// TwinCAT 3 PLC project OEF_1
// ProgramVersion: 3.1.4024.0
// libraries:
//   Tc2_Standard, * (Beckhoff Automation GmbH)
//   Tc2_System, * (Beckhoff Automation GmbH)
//   Tc3_Module, * (Beckhoff Automation GmbH)
// project tree:
//   / PlcTask.TcTTO
//   POUs/ MAIN.TcPOU
// real-time tasks:
//   TASK PlcTask: cycle T#10ms, priority 20, ADS port 350
//   TASK PlcTask1: cycle T#10ms, priority 21, ADS port 351
//   TASK PlcTask2: cycle T#10ms, priority 22, ADS port 352
//   TASK PlcTask3: cycle T#10ms, priority 23, ADS port 353
//   TASK PlcTask4: cycle T#10ms, priority 24, ADS port 354
//   TASK PlcTask5: cycle T#10ms, priority 25, ADS port 355
//   TASK PlcTask6: cycle T#10ms, priority 26, ADS port 356
// I/O:
//   DEVICE Device 1 (EtherCAT), AmsNetId 5.59.222.235.2.1
//     Term 1 (EK1200) [EK1200-5000 EtherCAT Power supply (2A E-Bus)]
//       Term 2 (EL1008) [EL1008 8Ch. Dig. Input 24V, 3ms]
//       Term 3 (EL2008) [EL2008 8Ch. Dig. Output 24V, 0.5A]
//       Term 4 (EL3062) [EL3062 2Ch. Ana. Input 0-10V]
//       Term 5 (EL4002) [EL4002 2Ch. Ana. Output 0-10V, 12bit]
//       Term 6 (EL1904) [EL1904, 4 Ch. Safety Input 24V, TwinSAFE]
//         modules: Module 1 (FSOES)
//       Term 7 (EL6900) [EL6900, TwinSAFE PLC]
//       Term 8 (EL2904) [EL2904, 4 Ch. Safety Output 24V, 0.5A, TwinSAFE]
//         modules: Module 1 (FSOES), Module 2 (DO)
//       Term 9 (EK1110) [EK1110 EtherCAT extension]
// variable links:
//   OEF_4/OEF_4 Instance <-> Device 1 (EtherCAT)/Term 1 (EK1200)/Term 2 (EL1008)
//     PlcTask Inputs/MAIN.bKnop <-> Channel 1/Input
//   OEF_4/OEF_4 Instance <-> Device 1 (EtherCAT)/Term 1 (EK1200)/Term 3 (EL2008)
//     PlcTask Outputs/MAIN.bLED1 <-> Channel 1/Output
//   OEF_5/OEF_5 Instance <-> Device 1 (EtherCAT)/Term 1 (EK1200)/Term 3 (EL2008)
//     PlcTask Outputs/MAIN.bLED1 <-> Channel 2/Output
//   OEF_6/OEF_6 Instance <-> Device 1 (EtherCAT)/Term 1 (EK1200)/Term 3 (EL2008)
//     PlcTask Outputs/MAIN.bLED1 <-> Channel 3/Output

CONFIGURATION OEF_1
    RESOURCE PLC ON TwinCAT3
        TASK PlcTask(INTERVAL := T#10ms, PRIORITY := 20);
        PROGRAM MAIN WITH PlcTask : MAIN;
    END_RESOURCE
END_CONFIGURATION

// ---- POUs/MAIN.TcPOU
PROGRAM MAIN
VAR

	fbKeuken: TP := (PT := TIME#60ms);
	bKeuken AT %i*: BOOL := false;
	bLED1 AT %Q*: BOOL := false;
END_VAR

fbKeuken(IN:= bKeuken , Q=>bLED1);

END_PROGRAM
